TYPE OutputBase_10CEE7DE :
STRUCT
END_STRUCT
END_TYPE

(* stored: Version 1.1.0.1, ProductVersion 3.1.4024.9
   DUT OutputBase_10CEE7DE: Id {1f43c418-f421-04d8-3ca4-1b77ba7ed728} *)
